INTERFACE I_AsyncRpcCallQueue

METHOD PUBLIC TryAddRpcCall : BOOL
VAR_INPUT
	CallingParameters : I_Deserializer;
	CallingAsynchronousRpcResponse : I_AsynchronousRpcResponse;
	CallingHandler : I_AsynchronousRpcHandler;
END_VAR
END_METHOD

END_INTERFACE

(* stored: Version 1.1.0.1, ProductVersion 3.1.4026.13
   Itf I_AsyncRpcCallQueue: Id {1f61c9cb-5ed5-06a5-1cb6-e63faa3bd4a9}
   Method TryAddRpcCall: Id {30ee6558-a303-04e7-0846-f4c30c270ab6} *)
